{attribute 'qualified_only'}
{attribute 'strict'}
{attribute 'to_string'}
TYPE L_Attenuators :
(
    AT1L0 := 1, // FEE Combo Gas/Solid Attenuator
    AT2L0 := 2 // FEE Solid Attenuator
);
END_TYPE

(* stored: Version 1.1.0.1
   DUT L_Attenuators: Id {fbbe85ee-383c-4931-afa7-af2367ddc0a1} *)
